FUNCTION_BLOCK fb_MessageDataCtrl EXTENDS fb_MessageData
VAR
  _stCtrl       : REFERENCE TO ST_MESSAGE_CTRL;
  _stState      : REFERENCE TO ST_MESSAGE_STATE;

  _eCmd,
  _eCmdOld      : E_MESSAGE_CTRL;

  _eResult,
  _eJobResult   : E_PROGRESS;

  _eState       : E_MESSAGE_STATE;

END_VAR

//-----------------------------------------------------------------------------
// check pointers
//-----------------------------------------------------------------------------
IF NOT Check()
THEN
  _eResult                      := E_PROGRESS.PROGRESS_ERROR;
  RETURN;
END_IF
//-----------------------------------------------------------------------------
// check date
// new message file for a new day
//-----------------------------------------------------------------------------
IF (FolderDate(_dtLocalTime) <> _sFolderDate)
THEN
  _bFileCreated                 := FALSE;
END_IF
//-----------------------------------------------------------------------------
//----------------------------------------------------------------------------- 
// copy to local for debug
_eCmd                         := _stCtrl.Cmd;

// cyclic check for command change
// get state for cmd
IF (_eCmd <> _eCmdOld)
THEN
  // get matching sdtate for Ctrl.Cmd
  _eState                     := Cmd(_eCmd);
  _eCmdOld                    := _eCmd;
END_IF


CASE _eResult
OF
  E_PROGRESS.PROGRESS_INVALID:
    _stState.State            := E_MESSAGE_STATE.MSG_STATE_NULL;

  E_PROGRESS.PROGRESS_ERROR:
    _stState.State            := _eState + E_PROGRESS.PROGRESS_ERROR;

  E_PROGRESS.PROGRESS_DONE:
    _stState.State            := _eState + E_PROGRESS.PROGRESS_DONE;

ELSE
  // work in progress
  // update progress for extern use
  _stState.State              := _eState + _eResult;

  CASE _eState
  OF
    E_MESSAGE_STATE.MSG_STATE_INIT:
      _eResult                := BuildFolder(TRUE);


    E_MESSAGE_STATE.MSG_STATE_IDLE:
      IF (_nMsgIndex < GVL_MSG.MAX_MESSAGE - GVL_MSG.MAX_MESSAGE/10)
      THEN
        _eResult              := E_PROGRESS.PROGRESS_WORKING;
      ELSE
        _eResult              := E_PROGRESS.PROGRESS_DONE;
        _nMsgIndex            := 0;
        // copy from attached list to local
        memcpy(ADR(_aWriteList), _pMsgList, SIZEOF(_aWriteList));
        // clear attached list
        memset(_pMsgList, 0, SIZEOF(_aWriteList));
      END_IF


    E_MESSAGE_STATE.MSG_STATE_WRITE:
      _eResult                := BuildFileData(TRUE);

  ELSE
      _eResult               := E_PROGRESS.PROGRESS_INVALID;
  END_CASE
END_CASE

METHOD BuildFileData : e_progress
VAR_INPUT
  Execute     : BOOL;
END_VAR
VAR_INST
  _nErrorId   : UDINT;
  _eState,
  _eRes       : E_PROGRESS;
  _eFlow      : E_MESSAGE_FLOW;

  _nStringLength  : UINT;
END_VAR
//-----------------------------------------------------------------------------
IF NOT Execute 
THEN
  _eRes                           := WriteData(FALSE);
  _eRes                           := BuildFolder(FALSE);
	_eState                         := E_PROGRESS.PROGRESS_INIT; 
END_IF 
//-----------------------------------------------------------------------------
IF NOT Check() 
THEN 
	BuildFileData                   := E_PROGRESS.PROGRESS_ERROR; 
	RETURN; 
END_IF
//-----------------------------------------------------------------------------
//-----------------------------------------------------------------------------
CASE _eState
OF
  E_PROGRESS.PROGRESS_INIT:
    IF Execute
    THEN
      _nErrorId                   := 0;
      _iStart 	                  := 1;
      _iEnd 		                  := SEL((_nMsgIndex > GVL_MSG.MAX_MESSAGE-1),
                                          _nMsgIndex,
                                          GVL_MSG.MAX_MESSAGE);

      memset(ADR(_sWriteData),0,SIZEOF(_sWriteData));

      IF (_sFolderDate <> FolderDate(_dtLocalTime))
      THEN
        _eState                   := E_PROGRESS.PROGRESS_PREPARE;
      ELSE
        _eState                   := E_PROGRESS.PROGRESS_BUSY;
        _eFlow                    := E_MESSAGE_FLOW.MSG_FLOW_LINE_START;
      END_IF
    END_IF
END_CASE
//-----------------------------------------------------------------------------
//-----------------------------------------------------------------------------
CASE _eState
OF
  E_PROGRESS.PROGRESS_PREPARE:
    _eRes                         := BuildFolder(TRUE);
    CASE _eRes
    OF
      E_PROGRESS.PROGRESS_DONE:
      _eState                     := E_PROGRESS.PROGRESS_BUSY;
      _eFlow                      := E_MESSAGE_FLOW.MSG_FLOW_LINE_START;

      E_PROGRESS.PROGRESS_ERROR:
      _eState                     := E_PROGRESS.PROGRESS_ERROR;
    END_CASE
END_CASE
//-----------------------------------------------------------------------------
//-----------------------------------------------------------------------------
CASE _eState
OF
  E_PROGRESS.PROGRESS_BUSY:
  CASE _eFlow
  OF
    E_MESSAGE_FLOW.MSG_FLOW_LINE_START:
      _eRes                       := BuildFolder(FALSE);
      _nErrIndex                  := 0; // rise and shine, all quarrels erased but not forgotten
      _nMsgIndex                  := 0;
  
      // copy from attached list to local
      memcpy(ADR(_aWriteList), _pMsgList, SIZEOF(_aWriteList));
  
      // clear attached list
      memset(_pMsgList, 0, SIZEOF(_aWriteList));


      _eFlow                      := E_MESSAGE_FLOW.MSG_FLOW_LINE_BUILD;
      _iCount                     := _iStart;
  END_CASE
  CASE _eFlow
  OF
    E_MESSAGE_FLOW.MSG_FLOW_LINE_BUILD:
      _eFlow                      := E_MESSAGE_FLOW.MSG_FLOW_LINE_CHECK;
      IF (_aWriteList[_iCount].eType > E_MessageType.eMessageEmpty)
      THEN
        _sTmp                     := TO_STRING(_aWriteList[_iCount].eType);
        _sTmp                     := Tc2_Standard.CONCAT(_sTmp, _sTab);
        _sTmp                     := Tc2_Standard.CONCAT(_sTmp, _aWriteList[_iCount].tTime);
        _sTmp                     := Tc2_Standard.CONCAT(_sTmp, _sTab);
        _sTmp                     := Tc2_Standard.CONCAT(_sTmp, Device_To_String(_aWriteList[_iCount].eDevice));
        _sTmp                     := Tc2_Standard.CONCAT(_sTmp, _sTab);
        _sTmp                     := Tc2_Standard.CONCAT(_sTmp, TO_STRING(_aWriteList[_iCount].eSubdevice));
        _sTmp                     := Tc2_Standard.CONCAT(_sTmp, _sTab);
        _sTmp                     := Tc2_Standard.CONCAT(_sTmp, TO_STRING(_aWriteList[_iCount].iErrorNumber));
        _sTmp                     := Tc2_Standard.CONCAT(_sTmp, _sTab);
        _sTmp                     := Tc2_Standard.CONCAT(_sTmp, _aWriteList[_iCount].sText);
        _sTmp                     := Tc2_Standard.CONCAT(_sTmp, _sNewLine);
        Builder(ADR(_sTmp), ADR(_sWriteData), StringLen(ADR(_sTmp)));
      END_IF
      _iCount                     := _iCount + 1;
  END_CASE
  CASE _eFlow
  OF
    E_MESSAGE_FLOW.MSG_FLOW_LINE_CHECK:
    IF NOT (_iCount > _iEnd)
    THEN
      _eFlow                      := E_MESSAGE_FLOW.MSG_FLOW_LINE_BUILD;
    ELSE
      _eState                     := E_PROGRESS.PROGRESS_WORKING;
      _eFlow                      := E_MESSAGE_FLOW.MSG_FLOW_WRITE_FILE_BUSY;
    END_IF
  END_CASE
END_CASE
//-----------------------------------------------------------------------------
//-----------------------------------------------------------------------------
CASE _eState
OF
  E_PROGRESS.PROGRESS_WORKING:
  CASE _eFlow
  OF
    E_MESSAGE_FLOW.MSG_FLOW_WRITE_FILE_BUSY:
      _nStringLength              := StringLen(ADR(_sWriteData));
      IF NOT (_nStringLength > 1)
      THEN
        _eState                   := E_PROGRESS.PROGRESS_DONE; 
       _eFlow                     := E_MESSAGE_FLOW.MSG_FLOW_WRITE_FILE_DONE;
      ELSE
        _eFlow                    := E_MESSAGE_FLOW.MSG_FLOW_WRITE_FILE_END;
        _eRes                     := WriteData(FALSE);
      END_IF
  END_CASE
  CASE _eFlow
  OF
    E_MESSAGE_FLOW.MSG_FLOW_WRITE_FILE_END:
      _eRes                       := WriteData(TRUE);

      IF (_eRes = E_PROGRESS.PROGRESS_ERROR)
      THEN
        _eState                   := E_PROGRESS.PROGRESS_ERROR;

      ELSIF (_eRes = E_PROGRESS.PROGRESS_DONE)
      THEN
        _eState                   := E_PROGRESS.PROGRESS_DONE;
        _eFlow                    := E_MESSAGE_FLOW.MSG_FLOW_WRITE_FILE_DONE;
        _eRes                     := WriteData(FALSE);
      END_IF
  END_CASE
END_CASE
//-----------------------------------------------------------------------------
//-----------------------------------------------------------------------------

BuildFileData                     := _eState;
END_METHOD

METHOD BuildFolder : e_progress
VAR_INPUT
  Execute           : BOOL;
END_VAR
VAR_INST
  _nErrorId   : UDINT;
  _eState     : E_PROGRESS;
  _eFlow      : E_MESSAGE_FLOW;
END_VAR
//-----------------------------------------------------------------------------
IF NOT Execute 
THEN 
	_eState                       := E_PROGRESS.PROGRESS_INIT; 
END_IF 
//-----------------------------------------------------------------------------
IF NOT Check() 
THEN 
	BuildFolder                   := E_PROGRESS.PROGRESS_ERROR; 
	RETURN; 
END_IF
//-----------------------------------------------------------------------------
//-----------------------------------------------------------------------------
CASE _eState
OF
  E_PROGRESS.PROGRESS_INIT:
    IF Execute
    THEN
      _nErrorId                 := 0;
      _bFileCreated             := FALSE;

      _sFolderDate              := FolderDate(_dtLocalTime);
      _eState                   := E_PROGRESS.PROGRESS_BUSY;
      _eFlow                    := E_MESSAGE_FLOW.MSG_FLOW_ROOT;
    END_IF
END_CASE
//-----------------------------------------------------------------------------
//-----------------------------------------------------------------------------
CASE _eState
OF
  E_PROGRESS.PROGRESS_BUSY:
  CASE _eFlow
  OF
    E_MESSAGE_FLOW.MSG_FLOW_ROOT:
      _eFlow                    := E_MESSAGE_FLOW.MSG_FLOW_ROOT_CREATE;
      _fbCreateDir.sPathName    := left(_pDirRoot^,len(_pDirRoot^)-1);
      _fbCreateDir(
              bExecute	        := FALSE);
    
    E_MESSAGE_FLOW.MSG_FLOW_ROOT_CREATE:
      (* create root folder *)
      _fbCreateDir(
              bExecute	        := TRUE);
      IF _fbCreateDir.bBusy
      THEN
        _eFlow                  := E_MESSAGE_FLOW.MSG_FLOW_ROOT_CREATE_BUSY;
      END_IF
    
    E_MESSAGE_FLOW.MSG_FLOW_ROOT_CREATE_BUSY:
      _fbCreateDir(
              bExecute	        := TRUE);
      IF NOT _fbCreateDir.bBusy
      THEN
        _eState                 := E_PROGRESS.PROGRESS_PREPARE;
        _eFlow                  := E_MESSAGE_FLOW.MSG_FLOW_FOLDER;
      END_IF
  END_CASE
END_CASE
//-----------------------------------------------------------------------------
//-----------------------------------------------------------------------------
CASE _eState
OF
  E_PROGRESS.PROGRESS_PREPARE:
  CASE _eFlow
  OF
    E_MESSAGE_FLOW.MSG_FLOW_FOLDER:
      _eFlow                    := E_MESSAGE_FLOW.MSG_FLOW_FOLDER_CREATE;
      _sFolderDate              := FolderDate(_dtLocalTime);
      _fbCreateDir.sPathName    := concat(_pDirRoot^, _sFolderDate);
      _fbCreateDir(
              bExecute	        := FALSE);
  
    E_MESSAGE_FLOW.MSG_FLOW_FOLDER_CREATE:
      (* create active folder *)
      _fbCreateDir(
              bExecute	        := TRUE);
      IF _fbCreateDir.bBusy
      THEN
        _eFlow                  := E_MESSAGE_FLOW.MSG_FLOW_FOLDER_CREATE_BUSY;
      END_IF
    
    E_MESSAGE_FLOW.MSG_FLOW_FOLDER_CREATE_BUSY:
      _fbCreateDir(
              bExecute	        := TRUE);
      IF NOT _fbCreateDir.bBusy
      THEN
        _eState                 := E_PROGRESS.PROGRESS_CHECK;
        _eFlow                  := E_MESSAGE_FLOW.MSG_FLOW_FILE_CREATE_DONE;
        _fbCreateDir(
                bExecute	      := FALSE);
      END_IF
  END_CASE
END_CASE
//-----------------------------------------------------------------------------
//-----------------------------------------------------------------------------
CASE _eState
OF
  E_PROGRESS.PROGRESS_CHECK:
  CASE _eFlow
  OF
    E_MESSAGE_FLOW.MSG_FLOW_FILE_CREATE_DONE:
      _eState                   := E_PROGRESS.PROGRESS_DONE;
      _bFileCreated             := TRUE;

      // build complete file path
      _sTmp                     := concat(concat(_pFileRoot^, _sFolderDate),'.txt');
      _sTmp                     := concat('\', _sTmp);
      _sFilename                := concat(_fbCreateDir.sPathName, _sTmp);
  END_CASE
END_CASE

BuildFolder                     := _eState;
END_METHOD

METHOD Check : BOOL
VAR_INPUT
END_VAR

IF NOT __ISVALIDREF(_stCtrl)
THEN
  _eCheck       := E_MESSAGE_CHECK.POINTER_CTRL_INVALID;
  RETURN;
END_IF

IF NOT __ISVALIDREF(_stState)
THEN
  _eCheck       := E_MESSAGE_CHECK.POINTER_STATE_INVALID;
  RETURN;
END_IF
//-----------------------------------------------------------------
//-----------------------------------------------------------------
IF NOT (_dtLocalTime <> 0)
THEN
  _eCheck       := E_MESSAGE_CHECK.POINTER_TIME_INVALID;
  RETURN;
END_IF

IF NOT (_pMsgList <> 0)
THEN
  _eCheck       := E_MESSAGE_CHECK.POINTER_LIST_INVALID;
  RETURN;
END_IF

IF NOT (_pFileRoot <> 0)
THEN
  _eCheck       := E_MESSAGE_CHECK.POINTER_ROOT_FILE_INVALID;
  RETURN;
END_IF

IF NOT (_pDirRoot <> 0)
THEN
  _eCheck       := E_MESSAGE_CHECK.POINTER_ROOT_DIR_INVALID;
  RETURN;
END_IF

IF NOT __ISVALIDREF(_nMsgIndex)
THEN
  _eCheck       := E_MESSAGE_CHECK.POINTER_MSG_IDX_INVALID;
  RETURN;
END_IF

IF NOT __ISVALIDREF(_nErrIndex)
THEN
  _eCheck       := E_MESSAGE_CHECK.POINTER_ERR_IDX_INVALID;
  RETURN;
END_IF


_eCheck         := E_MESSAGE_CHECK.CHECK_DONE;
Check           := TRUE;
END_METHOD

METHOD Cmd : e_message_state
VAR_INPUT
  Command     : e_message_ctrl;
END_VAR


CASE Command
OF
  E_MESSAGE_CTRL.MSG_CTRL_NULL:
    _eResult                    := E_PROGRESS.PROGRESS_INVALID;
    Cmd                         := E_MESSAGE_STATE.MSG_STATE_NULL;

  E_MESSAGE_CTRL.MSG_CTRL_INIT:
    _eResult                    := BuildFolder(FALSE);
    Cmd                         := E_MESSAGE_STATE.MSG_STATE_INIT;

  E_MESSAGE_CTRL.MSG_CTRL_IDLE:
    _eResult                    := BuildFileData(FALSE);
    Cmd                         := E_MESSAGE_STATE.MSG_STATE_IDLE;

  E_MESSAGE_CTRL.MSG_CTRL_WRITE:
    _eResult                    := BuildFileData(FALSE);
    Cmd                         := E_MESSAGE_STATE.MSG_STATE_WRITE;
    IF (_nMsgIndex = 0)
    THEN
       // go back to sleep
      _eResult                := E_PROGRESS.PROGRESS_DONE;
    END_IF
ELSE
    //_eResult                    := E_PROGRESS.PROGRESS_ERROR;
    Cmd                         := E_MESSAGE_STATE.MSG_STATE_NULL;
END_CASE
END_METHOD

PROPERTY Ctrl : REFERENCE to ST_MESSAGE_CTRL
SET
_stCtrl ref= Ctrl;
END_SET
END_PROPERTY

PROPERTY FileCreated : bool
GET
FileCreated := _bFileCreated;
END_GET
END_PROPERTY

PROPERTY State : REFERENCE TO ST_MESSAGE_STATE
SET
_stState ref= State;
END_SET
END_PROPERTY

END_FUNCTION_BLOCK

(* stored: Version 1.1.0.1, ProductVersion 3.1.4026.13
   POU fb_MessageDataCtrl: Id {93d80d01-2f62-466c-9079-6d221a01cc61}, SpecialFunc None
   Folder methods: Id {7b7fb26d-2d9f-4358-abe4-81158e2934a0}
   Method BuildFileData: Id {f7ac25e2-99d5-4c0b-91cf-be66388bcc74}
   Method BuildFolder: Id {b9409663-b8f3-4d10-93b2-c286ad3fd28e}
   Method Check: Id {16d2b48d-131a-4d23-8d16-d64574df8817}
   Method Cmd: Id {1e20a8d5-c56d-4a13-9fd2-095411ce6509}
   Property Ctrl: Id {ad0b8e62-400b-4cb4-a754-b7b7d59451f1}
   Set Set: Id {95913b40-b2cc-4a27-bf6c-c8568a5955ad}
   Property FileCreated: Id {8e957e89-8bcc-4769-a2a5-0957dcd98f08}
   Get Get: Id {9a4d4de6-af54-40db-ae74-ad042e4d9799}
   Property State: Id {53cb4b2a-946d-480e-b295-5d17e7ee9c6b}
   Set Set: Id {0827ebbb-dde2-4a65-b760-bc69425f5977} *)
